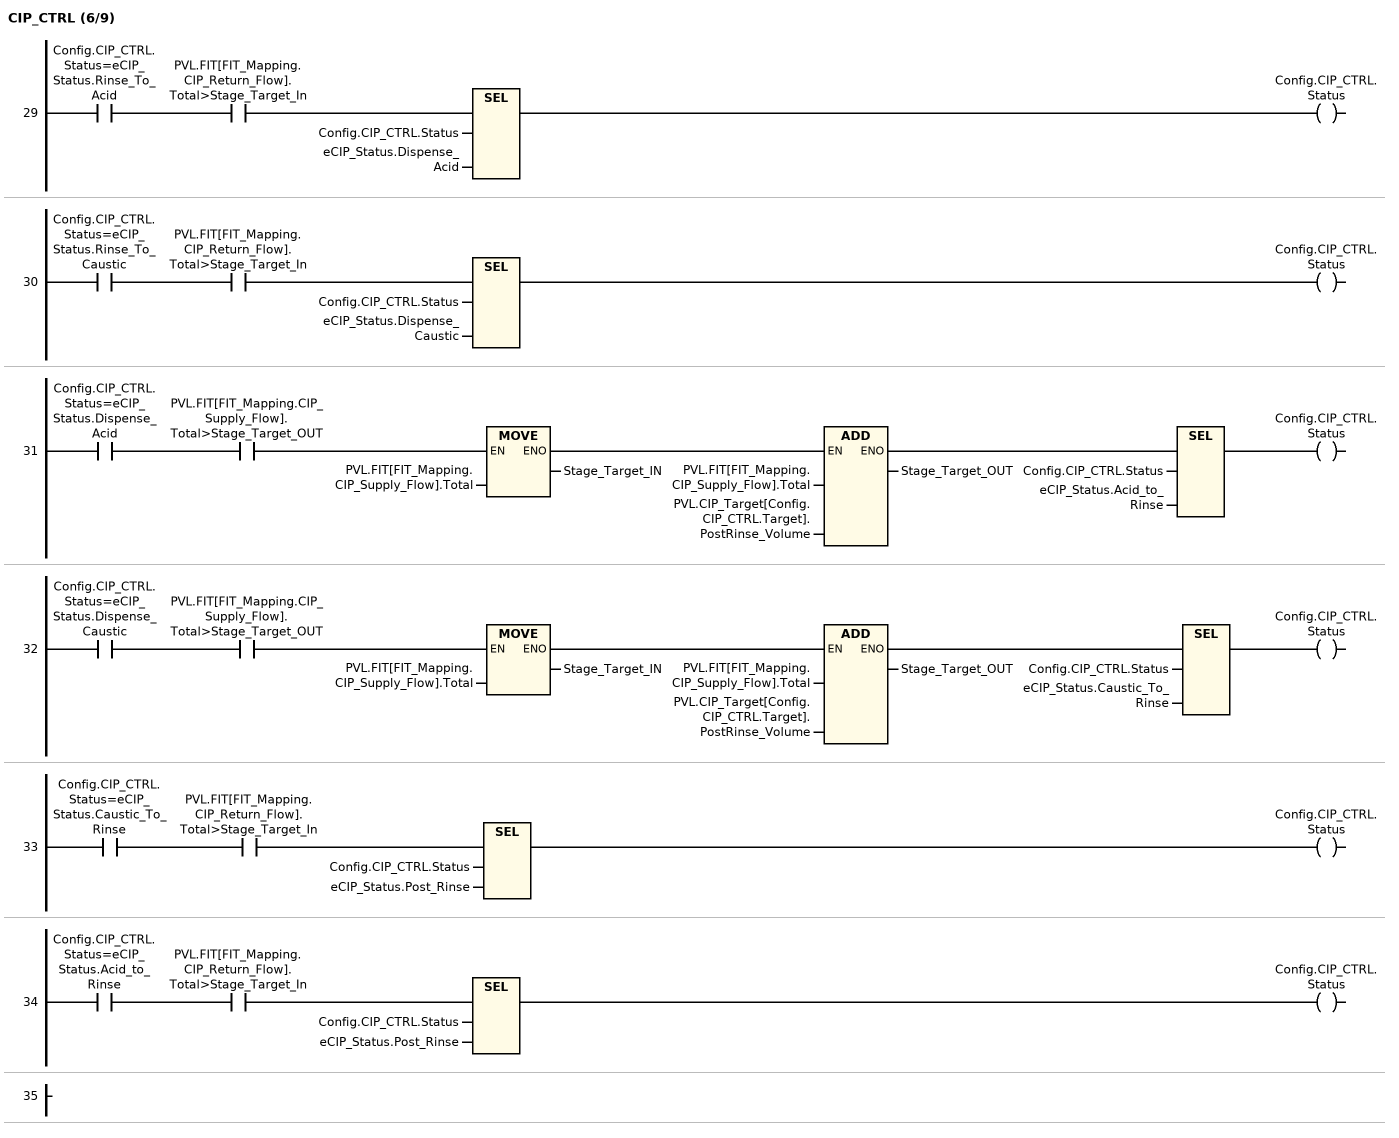
// NETWORK 29
Config.CIP_CTRL.Status := SEL((Config.CIP_CTRL.Status=eCIP_Status.Rinse_To_Acid) AND (PVL.FIT[FIT_Mapping.CIP_Return_Flow].Total>Stage_Target_In), Config.CIP_CTRL.Status, eCIP_Status.Dispense_Acid);

// NETWORK 30
Config.CIP_CTRL.Status := SEL((Config.CIP_CTRL.Status=eCIP_Status.Rinse_To_Caustic) AND (PVL.FIT[FIT_Mapping.CIP_Return_Flow].Total>Stage_Target_In), Config.CIP_CTRL.Status, eCIP_Status.Dispense_Caustic);

// NETWORK 31
_w16 := (Config.CIP_CTRL.Status=eCIP_Status.Dispense_Acid) AND (PVL.FIT[FIT_Mapping.CIP_Supply_Flow].Total>Stage_Target_OUT);
IF _w16 THEN Stage_Target_IN := PVL.FIT[FIT_Mapping.CIP_Supply_Flow].Total; END_IF
IF _w16 THEN
    Stage_Target_OUT := PVL.FIT[FIT_Mapping.CIP_Supply_Flow].Total + PVL.CIP_Target[Config.CIP_CTRL.Target].PostRinse_Volume;
END_IF
Config.CIP_CTRL.Status := SEL(_w16, Config.CIP_CTRL.Status, eCIP_Status.Acid_to_Rinse);

// NETWORK 32
_w17 := (Config.CIP_CTRL.Status=eCIP_Status.Dispense_Caustic) AND (PVL.FIT[FIT_Mapping.CIP_Supply_Flow].Total>Stage_Target_OUT);
IF _w17 THEN Stage_Target_IN := PVL.FIT[FIT_Mapping.CIP_Supply_Flow].Total; END_IF
IF _w17 THEN
    Stage_Target_OUT := PVL.FIT[FIT_Mapping.CIP_Supply_Flow].Total + PVL.CIP_Target[Config.CIP_CTRL.Target].PostRinse_Volume;
END_IF
Config.CIP_CTRL.Status := SEL(_w17, Config.CIP_CTRL.Status, eCIP_Status.Caustic_To_Rinse);

// NETWORK 33
Config.CIP_CTRL.Status := SEL((Config.CIP_CTRL.Status=eCIP_Status.Caustic_To_Rinse) AND (PVL.FIT[FIT_Mapping.CIP_Return_Flow].Total>Stage_Target_In), Config.CIP_CTRL.Status, eCIP_Status.Post_Rinse);

// NETWORK 34
Config.CIP_CTRL.Status := SEL((Config.CIP_CTRL.Status=eCIP_Status.Acid_to_Rinse) AND (PVL.FIT[FIT_Mapping.CIP_Return_Flow].Total>Stage_Target_In), Config.CIP_CTRL.Status, eCIP_Status.Post_Rinse);

// NETWORK 35

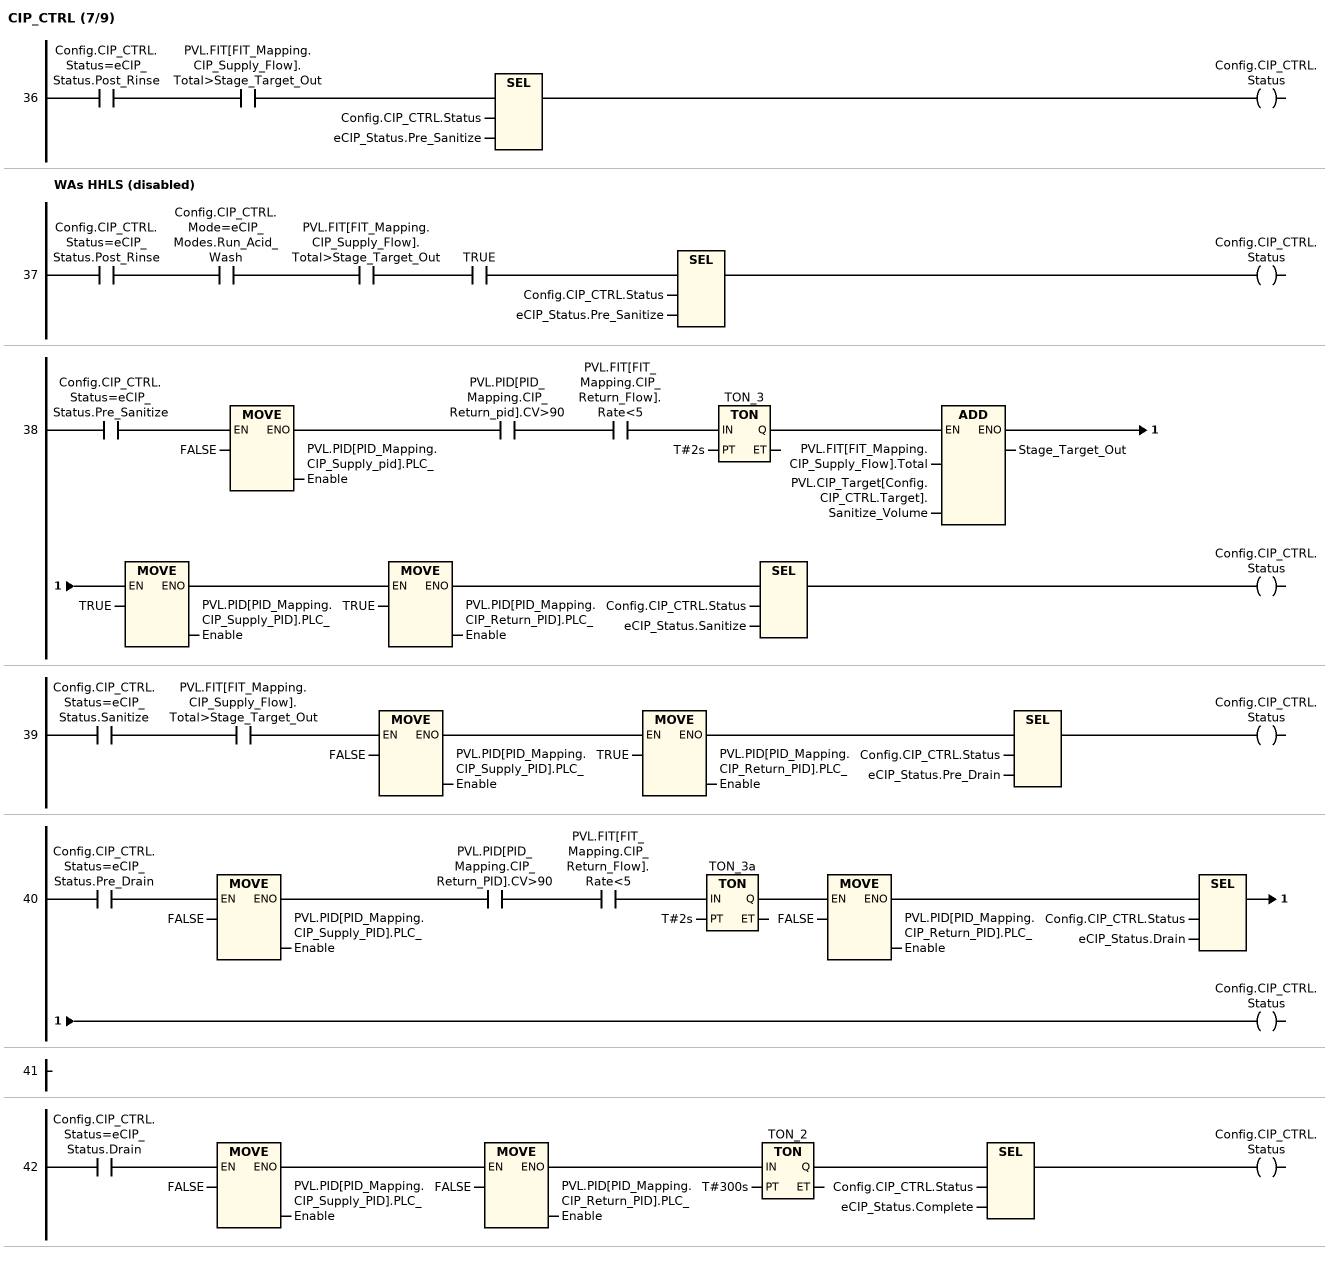
// NETWORK 36
Config.CIP_CTRL.Status := SEL((Config.CIP_CTRL.Status=eCIP_Status.Post_Rinse) AND (PVL.FIT[FIT_Mapping.CIP_Supply_Flow].Total>Stage_Target_Out), Config.CIP_CTRL.Status, eCIP_Status.Pre_Sanitize);

// NETWORK 37: WAs HHLS (disabled)
// Config.CIP_CTRL.Status := SEL(((Config.CIP_CTRL.Status=eCIP_Status.Post_Rinse) AND (Config.CIP_CTRL.Mode=eCIP_Modes.Run_Acid_Wash)) AND (PVL.FIT[FIT_Mapping.CIP_Supply_Flow].Total>Stage_Target_Out) AND TRUE, Config.CIP_CTRL.Status, eCIP_Status.Pre_Sanitize);

// NETWORK 38
_w18 := Config.CIP_CTRL.Status=eCIP_Status.Pre_Sanitize;
IF _w18 THEN PVL.PID[PID_Mapping.CIP_Supply_pid].PLC_Enable := FALSE; END_IF
TON_3(IN := _w18 AND (PVL.PID[PID_Mapping.CIP_Return_pid].CV>90) AND (PVL.FIT[FIT_Mapping.CIP_Return_Flow].Rate<5), PT := T#2s); // TON
_w19 := TON_3.Q;
IF _w19 THEN
    Stage_Target_Out := PVL.FIT[FIT_Mapping.CIP_Supply_Flow].Total + PVL.CIP_Target[Config.CIP_CTRL.Target].Sanitize_Volume;
END_IF
IF _w19 THEN PVL.PID[PID_Mapping.CIP_Supply_PID].PLC_Enable := TRUE; END_IF
IF _w19 THEN PVL.PID[PID_Mapping.CIP_Return_PID].PLC_Enable := TRUE; END_IF
Config.CIP_CTRL.Status := SEL(_w19, Config.CIP_CTRL.Status, eCIP_Status.Sanitize);

// NETWORK 39
_w20 := (Config.CIP_CTRL.Status=eCIP_Status.Sanitize) AND (PVL.FIT[FIT_Mapping.CIP_Supply_Flow].Total>Stage_Target_Out);
IF _w20 THEN PVL.PID[PID_Mapping.CIP_Supply_PID].PLC_Enable := FALSE; END_IF
IF _w20 THEN PVL.PID[PID_Mapping.CIP_Return_PID].PLC_Enable := TRUE; END_IF
Config.CIP_CTRL.Status := SEL(_w20, Config.CIP_CTRL.Status, eCIP_Status.Pre_Drain);

// NETWORK 40
_w21 := Config.CIP_CTRL.Status=eCIP_Status.Pre_Drain;
IF _w21 THEN PVL.PID[PID_Mapping.CIP_Supply_PID].PLC_Enable := FALSE; END_IF
TON_3a(IN := _w21 AND (PVL.PID[PID_Mapping.CIP_Return_PID].CV>90) AND (PVL.FIT[FIT_Mapping.CIP_Return_Flow].Rate<5), PT := T#2s); // TON
_w22 := TON_3a.Q;
IF _w22 THEN PVL.PID[PID_Mapping.CIP_Return_PID].PLC_Enable := FALSE; END_IF
Config.CIP_CTRL.Status := SEL(_w22, Config.CIP_CTRL.Status, eCIP_Status.Drain);

// NETWORK 41

// NETWORK 42
_w23 := Config.CIP_CTRL.Status=eCIP_Status.Drain;
IF _w23 THEN PVL.PID[PID_Mapping.CIP_Supply_PID].PLC_Enable := FALSE; END_IF
IF _w23 THEN PVL.PID[PID_Mapping.CIP_Return_PID].PLC_Enable := FALSE; END_IF
TON_2(IN := _w23, PT := T#300s); // TON
Config.CIP_CTRL.Status := SEL(TON_2.Q, Config.CIP_CTRL.Status, eCIP_Status.Complete);

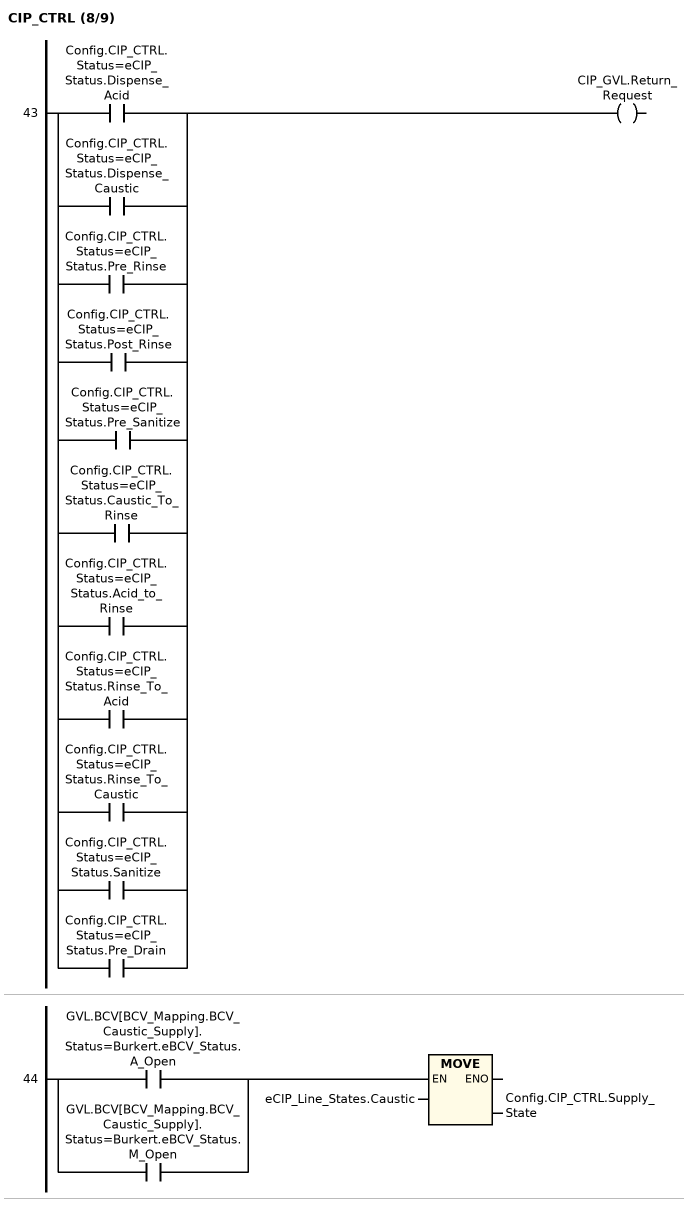
// NETWORK 43
CIP_GVL.Return_Request := (Config.CIP_CTRL.Status=eCIP_Status.Dispense_Acid) OR (Config.CIP_CTRL.Status=eCIP_Status.Dispense_Caustic) OR (Config.CIP_CTRL.Status=eCIP_Status.Pre_Rinse) OR (Config.CIP_CTRL.Status=eCIP_Status.Post_Rinse) OR (Config.CIP_CTRL.Status=eCIP_Status.Pre_Sanitize) OR (Config.CIP_CTRL.Status=eCIP_Status.Caustic_To_Rinse) OR (Config.CIP_CTRL.Status=eCIP_Status.Acid_to_Rinse) OR (Config.CIP_CTRL.Status=eCIP_Status.Rinse_To_Acid) OR (Config.CIP_CTRL.Status=eCIP_Status.Rinse_To_Caustic) OR (Config.CIP_CTRL.Status=eCIP_Status.Sanitize) OR (Config.CIP_CTRL.Status=eCIP_Status.Pre_Drain);

// NETWORK 44
IF (GVL.BCV[BCV_Mapping.BCV_Caustic_Supply].Status=Burkert.eBCV_Status.A_Open) OR (GVL.BCV[BCV_Mapping.BCV_Caustic_Supply].Status=Burkert.eBCV_Status.M_Open) THEN
    Config.CIP_CTRL.Supply_State := eCIP_Line_States.Caustic;
END_IF

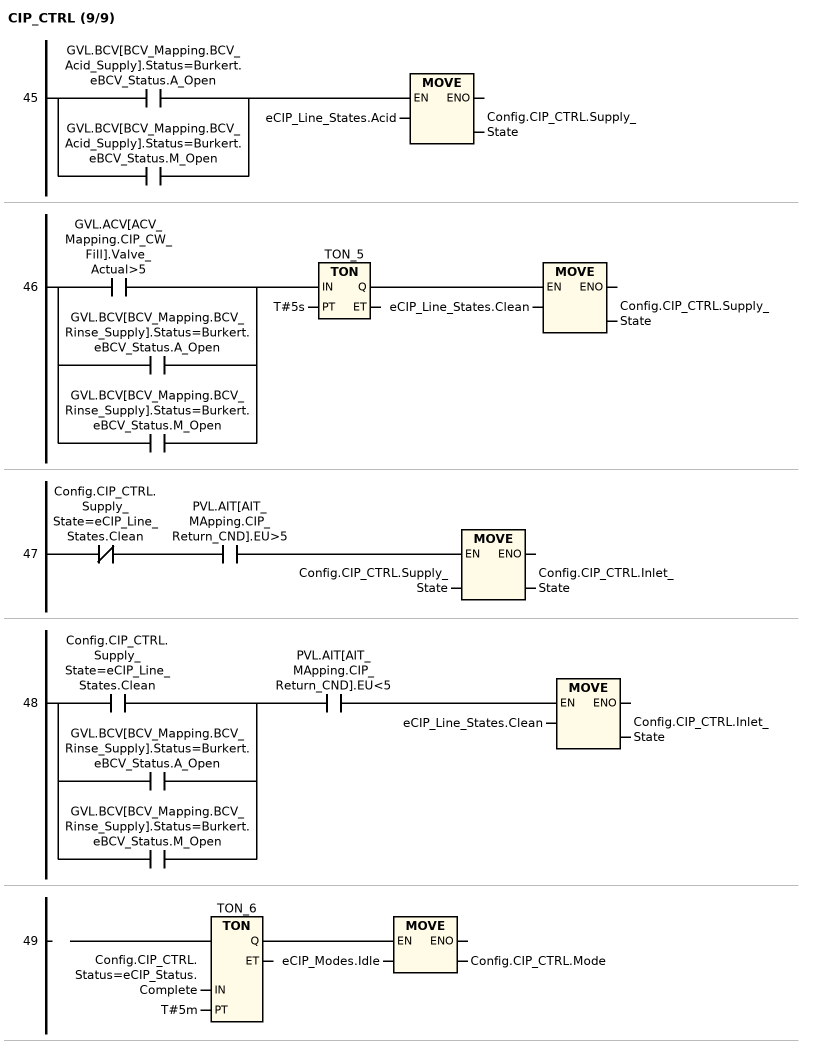
// NETWORK 45
IF (GVL.BCV[BCV_Mapping.BCV_Acid_Supply].Status=Burkert.eBCV_Status.A_Open) OR (GVL.BCV[BCV_Mapping.BCV_Acid_Supply].Status=Burkert.eBCV_Status.M_Open) THEN
    Config.CIP_CTRL.Supply_State := eCIP_Line_States.Acid;
END_IF

// NETWORK 46
TON_5(IN := (GVL.ACV[ACV_Mapping.CIP_CW_Fill].Valve_Actual>5) OR (GVL.BCV[BCV_Mapping.BCV_Rinse_Supply].Status=Burkert.eBCV_Status.A_Open) OR (GVL.BCV[BCV_Mapping.BCV_Rinse_Supply].Status=Burkert.eBCV_Status.M_Open), PT := T#5s); // TON
IF TON_5.Q THEN Config.CIP_CTRL.Supply_State := eCIP_Line_States.Clean; END_IF

// NETWORK 47
IF NOT (Config.CIP_CTRL.Supply_State=eCIP_Line_States.Clean) AND (PVL.AIT[AIT_MApping.CIP_Return_CND].EU>5) THEN
    Config.CIP_CTRL.Inlet_State := Config.CIP_CTRL.Supply_State;
END_IF

// NETWORK 48
IF ((Config.CIP_CTRL.Supply_State=eCIP_Line_States.Clean) OR (GVL.BCV[BCV_Mapping.BCV_Rinse_Supply].Status=Burkert.eBCV_Status.A_Open) OR (GVL.BCV[BCV_Mapping.BCV_Rinse_Supply].Status=Burkert.eBCV_Status.M_Open)) AND (PVL.AIT[AIT_MApping.CIP_Return_CND].EU<5) THEN
    Config.CIP_CTRL.Inlet_State := eCIP_Line_States.Clean;
END_IF

// NETWORK 49
TON_6(IN := Config.CIP_CTRL.Status=eCIP_Status.Complete, PT := T#5m); // TON
IF TON_6.Q THEN Config.CIP_CTRL.Mode := eCIP_Modes.Idle; END_IF

END_PROGRAM

// CIP_PID_CTRL
PROGRAM CIP_PID_CTRL
VAR
	
	R_TRIG_0: R_trig;
	F_TRIG_0: F_trig;
END_VAR
VAR // added by the converter: edge detectors and wires of the graphical bodies
    _w1, _w3, _w4, _w5, _w6, _w7, _w8, _w9 : ANY;
    _w2 : BOOL;
END_VAR

// HTX PID Loop
PVL.PID[PID_Mapping.CIP_HTX].PLC_Target := SEL(Config.CIP_CTRL.Mode=ecip_Modes.Idle, SEL(Config.CIP_CTRL.Status=eCip_Status.Sanitize, SEL((Config.CIP_CTRL.Status=eCip_Status.Acid_to_Rinse) OR (Config.CIP_CTRL.Status=eCip_Status.Caustic_To_Rinse) OR (Config.CIP_CTRL.Status=eCip_Status.Post_Rinse), SEL((Config.CIP_CTRL.Status=eCip_Status.Dispense_Acid) OR (Config.CIP_CTRL.Status=eCip_Status.Dispense_Caustic) OR (Config.CIP_CTRL.Status=eCip_Status.Rinse_To_Acid) OR (Config.CIP_CTRL.Status=eCip_Status.Rinse_To_Caustic) OR (Config.CIP_CTRL.Status=eCip_Status.Fill_Acid) OR (Config.CIP_CTRL.Status=eCip_Status.Fill_Caustic) OR False OR False OR (Config.CIP_CTRL.Status=eCip_Status.Low_Acid) OR (Config.CIP_CTRL.Status=eCip_Status.Low_Caustic), SEL((Config.CIP_CTRL.Status=eCip_Status.Fill_Rinse) OR False OR (Config.CIP_CTRL.Status=eCip_Status.line_charge) OR (Config.CIP_CTRL.Status=eCip_Status.Pre_Rinse), SEL((Config.CIP_CTRL.Status=eCip_Status.Heat_Acid) OR (Config.CIP_CTRL.Status=eCip_Status.Heat_Caustic) OR False, SEL(Config.CIP_CTRL.Status=eCip_Status.Heat_Rinse, PVL.PID[PID_Mapping.CIP_HTX].PLC_Target, PVL.CIP_Target[Config.CIP_CTRL.Target].PreRinse_Temp+5), PVL.CIP_Target[Config.CIP_CTRL.Target].Wash_Temp+5), PVL.CIP_Target[Config.CIP_CTRL.Target].PreRinse_Temp), PVL.CIP_Target[Config.CIP_CTRL.Target].Wash_Temp), PVL.CIP_Target[Config.CIP_CTRL.Target].PostRinse_Temp), PVL.CIP_Target[Config.CIP_CTRL.Target].Sanitize_Temp), PVL.PID[PID_Mapping.CIP_HTX].PLC_Target);
_w1 := NOT (Config.CIP_CTRL.Mode=ecip_Modes.Idle) AND (PVL.FIT[FIT_Mapping.CIP_Supply_Flow].Rate>5);
R_TRIG_0(CLK := _w1); // R_trig
F_TRIG_0(CLK := _w1); // F_trig
_w2 := SEL(R_TRIG_0.Q, SEL(F_TRIG_0.Q, PVL.PID[PID_Mapping.CIP_HTX].PLC_Enable, False), True);
PVL.PID[PID_Mapping.CIP_HTX].PLC_Enable := _w2;
IF _w2 THEN _w3 := PVL.PID[PID_Mapping.CIP_HTX].PLC_Target+5; END_IF
PVL.TT[TT_MApping.CIP_HTX_Discharge_Temp].Burkert.cAlarm_Config.Hi_Hi_Alarm := _w3;
PVL.TT[TT_MApping.CIP_Return_Temp].Burkert.cAlarm_Config.Hi_Hi_Alarm := _w3;
PVL.TT[TT_MApping.CIP_Acid_Temp].Burkert.cAlarm_Config.Hi_Hi_Alarm := _w3;
PVL.TT[TT_MApping.CIP_Caustic_Temp].Burkert.cAlarm_Config.Hi_Hi_Alarm := _w3;
IF _w2 THEN _w4 := PVL.PID[PID_Mapping.CIP_HTX].PLC_Target+2.5; END_IF
PVL.TT[TT_MApping.CIP_HTX_Discharge_Temp].Burkert.cAlarm_Config.Hi_Warn := _w4;
PVL.TT[TT_MApping.CIP_Return_Temp].Burkert.cAlarm_Config.Hi_Warn := _w4;
PVL.TT[TT_MApping.CIP_Acid_Temp].Burkert.cAlarm_Config.Hi_Warn := _w4;
PVL.TT[TT_MApping.CIP_Caustic_Temp].Burkert.cAlarm_Config.Hi_Warn := _w4;
IF _w2 THEN _w5 := PVL.PID[PID_Mapping.CIP_HTX].PLC_Target-2.5; END_IF
PVL.TT[TT_MApping.CIP_HTX_Discharge_Temp].Burkert.cAlarm_Config.Low_warn := _w5;
PVL.TT[TT_MApping.CIP_Return_Temp].Burkert.cAlarm_Config.Low_warn := _w5;
PVL.TT[TT_MApping.CIP_Acid_Temp].Burkert.cAlarm_Config.Low_warn := _w5;
PVL.TT[TT_MApping.CIP_Caustic_Temp].Burkert.cAlarm_Config.Low_warn := _w5;
IF _w2 THEN _w6 := PVL.PID[PID_Mapping.CIP_HTX].PLC_Target-5; END_IF
PVL.TT[TT_MApping.CIP_Return_Temp].Burkert.cAlarm_Config.Low_Low_Alarm := _w6;
PVL.TT[TT_MApping.CIP_HTX_Discharge_Temp].Burkert.cAlarm_Config.Low_Low_Alarm := _w6;
PVL.TT[TT_MApping.CIP_Acid_Temp].Burkert.cAlarm_Config.Low_Low_Alarm := _w6;
PVL.TT[TT_MApping.CIP_Caustic_Temp].Burkert.cAlarm_Config.Low_Low_Alarm := _w6;
_w7 := (Config.CIP_CTRL.Status=eCIP_Status.Dispense_Acid) OR (Config.CIP_CTRL.Status=eCIP_Status.Dispense_Caustic) OR (Config.CIP_CTRL.Status=eCIP_Status.line_charge) OR (Config.CIP_CTRL.Status=eCIP_Status.Post_Rinse) OR (Config.CIP_CTRL.Status=eCIP_Status.Pre_Sanitize) OR (Config.CIP_CTRL.Status=eCIP_Status.Sanitize) OR (Config.CIP_CTRL.Status=eCIP_Status.Caustic_To_Rinse) OR (Config.CIP_CTRL.Status=eCIP_Status.Acid_to_Rinse) OR (Config.CIP_CTRL.Status=eCIP_Status.Rinse_To_Acid) OR (Config.CIP_CTRL.Status=eCIP_Status.Rinse_To_Caustic) OR (Config.CIP_CTRL.Status=eCIP_Status.Pre_Drain) OR (Config.CIP_CTRL.Status=eCIP_Status.Pre_Rinse);
IF _w7 THEN _w8 := PVL.CIP_Target[Config.CIP_CTRL.Target].Rate; END_IF
PVL.PID[PID_Mapping.CIP_Supply_PID].PLC_Target := _w8;
IF _w7 THEN _w9 := SEL((Config.CIP_CTRL.Status=eCIP_Status.Pre_Sanitize) OR (Config.CIP_CTRL.Status=eCIP_Status.Pre_Drain), PVL.PID[PID_Mapping.CIP_Supply_PID].Actual, PVL.CIP_Target[Config.CIP_CTRL.Target].Rate); END_IF
PVL.PID[PID_Mapping.CIP_Return_PID].PLC_Target := _w9;

END_PROGRAM

// CIP_Valve_CTRL
PROGRAM CIP_Valve_CTRL
VAR

	F_TRIG_0: F_trig;
	R_TRIG_0: R_trig;
	TOF_0: TOF;
	TOF_1: TOF;
	TOF_2: TOF;
	Valve_Close_Delay:Time:=T#1s;
	TOF_3: TOF;
	TOF_4: TOF;
	TOF_5: TOF;
	TOF_6: TOF;
	TOF_7: TOF;
	TOF_8: TOF;
	TOF_9: TOF;
	TOF_10: TOF;
	MixProof_Index: INT;
	TOF_11: TOF;
	TON_0: TOn;
	TOF_7b: TOF;
	GEN_PULSE_0: BURKERT_OSCAT_BASIC.GEN_PULSE;
	Rinse_return_to_Drain:Bool;
END_VAR
VAR // added by the converter: edge detectors and wires of the graphical bodies
    _w1, _w2, _w3 : ANY;
END_VAR

_w1 := (Config.CIP_CTRL.Status=eCip_Status.Fill_Acid) OR (Config.CIP_CTRL.Status=eCip_Status.Fill_Caustic) OR (Config.CIP_CTRL.Status=eCip_Status.Fill_Rinse) OR (Config.CIP_CTRL.Status=eCIP_Status.line_charge) AND (GVL.LS[LS_Mapping.CIP_Rinse_HHLS].Status=DI_Status.Normal_Signal_OFF) OR (Config.CIP_CTRL.Status=eCIP_Status.Post_Rinse) OR (Config.CIP_CTRL.Status=eCIP_Status.Sanitize) OR (Config.CIP_CTRL.Status=eCIP_Status.Caustic_To_Rinse) OR (Config.CIP_CTRL.Status=eCIP_Status.Acid_to_Rinse);
GVL.ACV[ACV_Mapping.CIP_CW_Fill].PLC_CMD := SEL(_w1, 0.0, PVL.PID[PID_Mapping.CIP_Supply_PID].CV);
TOF_0(IN := _w1, PT := Valve_Close_Delay); // TOF
TOF_1(IN := (Config.CIP_CTRL.Status=eCip_Status.Fill_Acid) OR (Config.CIP_CTRL.Status=eCip_Status.Fill_Rinse) OR (Config.CIP_CTRL.Status=eCip_Status.Heat_Acid) OR (Config.CIP_CTRL.Status=eCip_Status.Heat_Rinse) OR (Config.CIP_CTRL.Status=eCip_Status.Fill_Caustic) OR (Config.CIP_CTRL.Status=eCip_Status.Heat_Caustic) OR (Config.CIP_CTRL.Status=eCip_Status.Low_Acid) OR (Config.CIP_CTRL.Status=eCip_Status.Low_Caustic), PT := Valve_Close_Delay); // TOF
gvl.BCV[bcv_mapping.BCV_CIP_Recirc].PLC_CMD := TOF_1.Q;
TOF_2(IN := ((Config.CIP_CTRL.Status=eCip_Status.Fill_Acid) OR (Config.CIP_CTRL.Status=eCip_Status.Heat_Acid) OR (Config.CIP_CTRL.Status=eCIP_Status.Dispense_Acid) OR (Config.CIP_CTRL.Status=eCIP_Status.Low_Acid) OR (Config.CIP_CTRL.Status=eCip_Status.Acid_to_Rinse)) AND NOT (Config.CIP_CTRL.Supply_State=eCIP_Line_States.Caustic), PT := Valve_Close_Delay); // TOF
gvl.BCV[bcv_mapping.BCV_acid_Return].PLC_CMD := TOF_2.Q;
TOF_3(IN := ((Config.CIP_CTRL.Status=eCip_Status.Fill_Caustic) OR (Config.CIP_CTRL.Status=eCip_Status.Heat_Caustic) OR (Config.CIP_CTRL.Status=eCIP_Status.Dispense_Caustic) OR (Config.CIP_CTRL.Status=eCip_Status.Low_Caustic) OR (Config.CIP_CTRL.Status=eCip_Status.Caustic_To_Rinse)) AND NOT (Config.CIP_CTRL.Supply_State=eCIP_Line_States.Acid), PT := Valve_Close_Delay); // TOF
gvl.BCV[bcv_mapping.BCV_Caustic_Return].PLC_CMD := TOF_3.Q;
TOF_4(IN := ((Config.CIP_CTRL.Status=eCip_Status.Heat_Caustic) OR (Config.CIP_CTRL.Status=eCIP_Status.Dispense_Caustic) OR (Config.CIP_CTRL.Status=eCip_Status.Low_Caustic) OR (Config.CIP_CTRL.Status=eCIP_Status.Rinse_To_Caustic)) AND NOT (Config.CIP_CTRL.Supply_State=eCIP_Line_States.Acid), PT := Valve_Close_Delay); // TOF
gvl.BCV[bcv_mapping.BCV_Caustic_Supply].PLC_CMD := TOF_4.Q;
TOF_6(IN := ((Config.CIP_CTRL.Status=eCip_Status.Heat_Acid) OR (Config.CIP_CTRL.Status=eCIP_Status.Dispense_Acid) OR (Config.CIP_CTRL.Status=eCIP_Status.Low_Acid) OR (Config.CIP_CTRL.Status=eCIP_Status.Rinse_To_Acid)) AND NOT (Config.CIP_CTRL.Supply_State=eCIP_Line_States.Caustic), PT := Valve_Close_Delay); // TOF
gvl.BCV[bcv_mapping.BCV_Acid_Supply].PLC_CMD := TOF_6.Q;
TOF_7(IN := (Config.CIP_CTRL.Status=eCIP_Status.Dispense_Acid) AND (GVL.LS[LS_Mapping.CIP_Acid_HHLS].Status=DI_Status.ALARM_Signal_ACTIVE) AND False OR (GVL.BCV[BCV_Mapping.BCV_acid_Return].Status=Burkert.eBCV_Status.A_Open) AND (GVL.LS[LS_Mapping.CIP_Acid_HHLS].Status=DI_Status.ALARM_Signal_ACTIVE), PT := Valve_Close_Delay); // TOF
gvl.BCV[bcv_mapping.BCV_Acid_Drain].PLC_CMD := TOF_7.Q;
TOF_8(IN := (Config.CIP_CTRL.Status=eCip_Status.Heat_Rinse) OR (Config.CIP_CTRL.Status=eCIP_Status.line_charge) OR (Config.CIP_CTRL.Status=eCIP_Status.Pre_Rinse) OR False OR False, PT := Valve_Close_Delay); // TOF
gvl.BCV[bcv_mapping.BCV_Rinse_Supply].PLC_CMD := TOF_8.Q;
_w2 := (Config.CIP_CTRL.Status=eCip_Status.Fill_Rinse) OR (Config.CIP_CTRL.Status=eCip_Status.Heat_Rinse) AND (gvl.BCV[BCV_Mapping.BCV_Caustic_Return].Status=Burkert.eBCV_Status.A_Closed) AND (gvl.BCV[BCV_Mapping.BCV_Caustic_Supply].Status=Burkert.eBCV_Status.A_Closed) OR (Config.CIP_CTRL.Status=eCIP_Status.Pre_Rinse) OR (Config.CIP_CTRL.Status=eCIP_Status.Post_Rinse) OR (Config.CIP_CTRL.Status=eCIP_Status.Pre_Sanitize);
Rinse_Return_To_Drain := (GVL.LS[LS_Mapping.CIP_Rinse_HHLS].Status=DI_Status.ALARM_Signal_ACTIVE) AND _w2;
TOF_5(IN := _w2 AND (GVL.LS[LS_Mapping.CIP_Rinse_HHLS].Status=DI_Status.Normal_Signal_OFF), PT := Valve_Close_Delay); // TOF
gvl.BCV[bcv_mapping.BCV_Rinse_Return].PLC_CMD := TOF_5.Q;
TOF_10(IN := True AND False AND (GVL.BCV[BCV_Mapping.BCV_Rinse_Return].Status=Burkert.eBCV_Status.A_Open) OR (Config.CIP_CTRL.Status=eCip_Status.Dispense_Acid) OR (Config.CIP_CTRL.Status=eCip_Status.Dispense_Caustic), PT := Valve_Close_Delay); // TOF
GVL.BCV[BCV_Mapping.BCV_Rinse_Drain].PLC_CMD := TOF_10.Q;
TOF_9(IN := (Config.CIP_CTRL.Status=eCIP_Status.Dispense_Acid) OR (Config.CIP_CTRL.Status=eCIP_Status.Dispense_Caustic) OR (Config.CIP_CTRL.Status=eCIP_Status.line_charge) OR (Config.CIP_CTRL.Status=eCIP_Status.Post_Rinse) OR (Config.CIP_CTRL.Status=eCIP_Status.Pre_Rinse) OR (Config.CIP_CTRL.Status=eCIP_Status.Rinse_To_Acid) OR (Config.CIP_CTRL.Status=eCIP_Status.Rinse_To_Caustic) OR (Config.CIP_CTRL.Status=eCIP_Status.Caustic_To_Rinse) OR (Config.CIP_CTRL.Status=eCIP_Status.Acid_to_Rinse) OR (Config.CIP_CTRL.Status=eCIP_Status.Sanitize), PT := Valve_Close_Delay); // TOF
// Supply
GVL.BCV[BCV_Mapping.BCV_CIP_Discharge].PLC_CMD := TOF_9.Q;
TOF_7b(IN := (GVL.BCV[BCV_Mapping.BCV_Caustic_Return].Status=Burkert.eBCV_Status.A_Open) AND (GVL.LS[LS_Mapping.CIP_Caustic_HHLS].Status=DI_Status.ALARM_Signal_ACTIVE) OR False, PT := Valve_Close_Delay); // TOF
gvl.BCV[bcv_mapping.BCV_Caustic_Drain].PLC_CMD := TOF_7b.Q;
TOF_11(IN := (Config.CIP_CTRL.Status=eCIP_Status.Rinse_To_Acid) OR (Config.CIP_CTRL.Status=eCIP_Status.Rinse_To_Caustic) OR (Config.CIP_CTRL.Status=eCIP_Status.Sanitize) OR Rinse_Return_To_Drain OR (Config.CIP_CTRL.Status=eCIP_Status.Pre_Drain) OR False, PT := Valve_Close_Delay); // TOF
// Return to Drain
GVL.BCV[BCV_Mapping.BCV_CIP_Loop_Drain].PLC_CMD := TOF_11.Q;
MixProof_Index := (MixProof_index+1) MOD B8681_Mapping.MPV_999;
_w3 := (Config.CIP_CTRL.Status	=eCip_Status.Complete) OR (Config.CIP_CTRL.Status	=eCip_Status.Idle) OR (Config.CIP_CTRL.Mode=ecip_modes.Prepare_Acid_Wash) OR (Config.CIP_CTRL.Mode=ecip_modes.Prepare_Caustic_Wash);
TON_0(IN := _w3, PT := T#10s); // TOn
GVL.B8691[MixProof_Index].PLC_CMD := SEL(Config.CIP_CTRL.Status	=eCip_Status.Drain, SEL(_w3, PVL.CIP_MixProof_Config[Config.CIP_CTRL.Target].Dispense_MixProof_Modes[MixProof_Index], SEL(TON_0.Q, eB8691_Modes.Auto, GVL.B8691[MixProof_Index].PLC_CMD)), PVL.CIP_MixProof_Config[Config.CIP_CTRL.Target].Drain_MixProof_Modes[MixProof_Index]);
// Config.CIP_CTRL.Status=eCIP_Status.Pre_Sanitize: input not connected

END_PROGRAM

// CIP_Pump_CTRL
PROGRAM CIP_Pump_CTRL
VAR
	R_TRIG_0: R_trig;
	F_TRIG_0: F_trig;
	TP_0: TP;
	F_TRIG_1: F_trig;
	R_TRIG_1: R_trig;
	//Base_Pump_Rate_LPM:REAL:=15.2;
	//Target_Sanitize_Per_L:REAL:=0.003; //3 ml
	GEN_PULSE_1: BURKERT_OSCAT_BASIC.GEN_PULSE;
	Sanitize_Min_Pump_Time:REAL:=5;
	Sanitize_LPS: REAL;
	Sanitizer_Target_Rate: REAL;
	Sanitizer_Min_Volume: REAL;
	Santizer_Rest_Time: REAL;
	TON_0: TON;
	Santizer_Dispense_Volume:REAL;
	R_TRIG_2: R_trig;
	F_TRIG_2: F_Trig;
	Sanitizer_Target_Volume:REAL;
	Santizer_Total_Time:REAL;
	Sanitize_Duration: REAL;
	Pump_OFF_Time: REAL;
	TP_1: TP;
	TP_2: TP;
	TON_1: TON;
END_VAR
VAR // added by the converter: edge detectors and wires of the graphical bodies
    _w1, _w2, _w3, _w4, _w5, _w6, _w8, _w10, _w12, _w14, _w17 : ANY;
    _w7 : BOOL;
    _w9, _w11, _w13, _w15, _w16 : REAL;
END_VAR

